// TwinCAT 3 PLC project Untitled1
// ProgramVersion: 3.1.4024.0
// libraries:
//   Tc2_Standard, * (Beckhoff Automation GmbH)
//   Tc2_System, * (Beckhoff Automation GmbH)
//   Tc3_Module, * (Beckhoff Automation GmbH)
//   VisuSymbols,3.5.10.0,System
// project tree:
//   / GlobalTextList.TcGTLO, PlcTask.TcTTO, Visualisierungsmanager.TcVMO (not stored)
//   GVLs/ GVL.TcGVL
//   POUs/ FuelMeasurement.TcPOU, MAIN.TcPOU
//   VISUs/ Visualization.TcVIS
// real-time tasks:
//   TASK PlcTask: cycle T#10ms, priority 20, ADS port 350
// I/O:
//   DEVICE Gerät 2 (CX7000), AmsNetId 5.156.235.236.3.1
//     Klemme 1 (CX7028) [CX7028-0000-0121]
//       modules: Module 1 (DIO_2x), Module 2 (Empty Module), Module 3 (DIO_2x), Module 4 (Empty Module), Module 5 (DI_2x), Module 6 (Empty Module), Module 7 (DI_2x), Module 8 (Empty Module)
// variable links:
//   Untitled1/Untitled1 Instance <-> Device 2 (CX7000)/Term 1 (CX7028)
//     PlcTask Inputs/GVL.sensorN1 <-> Module 1 (DIO_2x)/DIO_2x Input Channel 1/Input
//     PlcTask Inputs/GVL.sensorN2 <-> Module 3 (DIO_2x)/DIO_2x Input Channel 1/Input
//     PlcTask Outputs/GVL.ValveN2 <-> Module 3 (DIO_2x)/DIO_2x Output Channel 1/Output
//     PlcTask Outputs/GVL.valveN1 <-> Module 1 (DIO_2x)/DIO_2x Output Channel 1/Output

CONFIGURATION Untitled1
    RESOURCE PLC ON TwinCAT3
        TASK PlcTask(INTERVAL := T#10ms, PRIORITY := 20);
        PROGRAM MAIN WITH PlcTask : MAIN;
    END_RESOURCE
END_CONFIGURATION

// ---- GVLs/GVL.TcGVL
{attribute 'qualified_only'}
VAR_GLOBAL
	
	sensorN1 AT %I* : BOOL ;
	sensorN2 AT %I* : BOOL ;
	
	valveN1 AT %Q* : BOOL;
	ValveN2 AT %Q* : BOOL;
	
	bStartMeasurement : BOOL := FALSE;
	
	
END_VAR

// ---- POUs/MAIN.TcPOU
PROGRAM MAIN
VAR
	iCounter AT %Q*		: DINT;

	FuelMeasurement1 : FuelMeasurement;
	recordedTime : TIME ;
	bMeasurementOngoing1 : BOOL;
	valveN1 : BOOL ;
	valveN2 : BOOL ;
	FuelVolumePerSec : REAL;
	bMeasurementDone1 : BOOL := FALSE;
	
	//bMeasurementOngoing2: BOOL := FALSE;
END_VAR

iCounter := iCounter + 1;



FuelMeasurement1(bFuelMeasurement := GVL.bStartMeasurement, valveN1 => GVL.valveN1,valveN2 => GVL.ValveN2 , timeElapsed => recordedTime, bEndFB => bMeasurementDone1, FuelVolumePerSec => FuelVolumePerSec);

END_PROGRAM

// ---- POUs/FuelMeasurement.TcPOU
FUNCTION_BLOCK FuelMeasurement
VAR CONSTANT
	TankVolume : INT := 334; // The volume may vary depending on the tank volume.
	
END_VAR
VAR_INPUT
	bFuelMeasurement : BOOL := TRUE;
	
END_VAR
VAR_OUTPUT
	timeElapsed: TIME := T#0S;
	
	valveN1 : BOOL := FALSE;
	valveN2 : BOOL := FALSE;
	bEndFB : BOOL;
	FuelVolumePerSec : REAL := 0;
	
END_VAR
VAR
	bMeasurementDone : BOOL;
	readyToCount : BOOL := FALSE;
	timeStart: TIME;  
 	timerRunning: BOOL := FALSE;
	
	readyToClose : BOOL := FALSE;
	
	TimeToReal : REAL;
	//bMeasurementDone: BOOL := FALSE;
	INT1: INT :=0;
END_VAR

(*
IF GVL.sensorN1 AND GVL.sensorN2 AND bFuelMeasurement THEN
	valveN1 := TRUE;
	valveN2 := TRUE;
	readyToCount := TRUE;
END_IF  

IF NOT GVL.sensorN1 AND readyToCount THEN
	timeStart := TIME();
	readyToCount := FALSE;
	timerRunning := TRUE;
END_IF

IF NOT GVL.sensorN2 AND timerRunning THEN
	timeElapsed := TIME() - timeStart;
	timerRunning := FALSE;
	bMeasurementDone := TRUE;
END_IF

TimeToReal := (TIME_TO_REAL(timeElapsed)/ 1000); // The unit of TimeToReal is Second.
FuelVolumePerSec := TankVolume / (TimeToReal/60) ;

IF bMeasurementDone THEN
	valveN1 := FALSE;
	valveN2 := FALSE;
	bEndFB := TRUE;
END_IF
*)
(*--------------------State---------------------*)

CASE INT1 OF
0:
	IF GVL.sensorN1 AND GVL.sensorN2 THEN
		INT1 := 10;
	END_IF
10:  //Ready
	IF GVL.sensorN1 AND GVL.sensorN2 AND bFuelMeasurement THEN
	valveN1 := TRUE;
	valveN2 := TRUE;
	//readyToCount := TRUE;
	INT1 := 20;
	END_IF  
20:  //Wait for upper sensor
	IF NOT GVL.sensorN1 THEN
	timeStart := TIME();
	//readyToCount := FALSE;
	timerRunning := TRUE;
	INT1 := 30;
	END_IF   
30: //Wait for lower sensor
	IF NOT GVL.sensorN2 THEN
	timeElapsed := TIME() - timeStart;
	timerRunning := FALSE;
	//bMeasurementDone := TRUE;
	
	TimeToReal := (TIME_TO_REAL(timeElapsed)/ 1000); // The unit of TimeToReal is Second.
	FuelVolumePerSec := TankVolume / (TimeToReal/60) ;

	INT1 := 40;
	END_IF
40: //Measurement finished
	
	//IF bMeasurementDone THEN
	valveN1 := FALSE;
	valveN2 := FALSE;
	bEndFB := TRUE;
	//bMeasurementDone := FALSE;
	IF GVL.sensorN1 AND GVL.sensorN2 THEN
	INT1 := 10;
	END_IF
	
END_CASE;

END_FUNCTION_BLOCK

// ---- GlobalTextList.TcGTLO
TEXTLIST GlobalTextList
  158 = '%.2f ml/min'
  333 = '%0.1f'
  71 = 'Screen one'
  77 = 'State: %d'
END_TEXTLIST

// ---- VISUs/Visualization.TcVIS
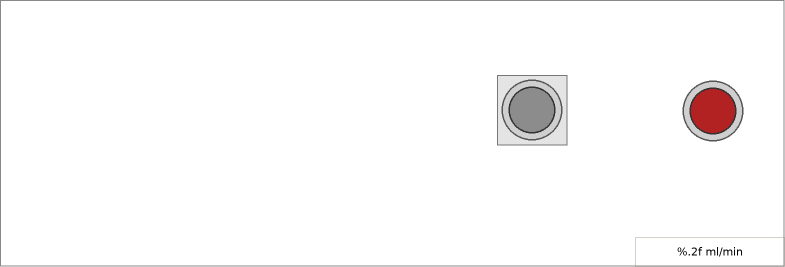
VISUALIZATION Visualization  // 785x267
    Lamp1 (678,76 70x70), variable: MAIN.FuelMeasurement1.timerRunning, style: Lamp-Lamp1-Red
    Textfield (635,237 150x30), "%.2f ml/min", text variable: MAIN.FuelVolumePerSec
    PushSwitch (497,75 70x70), variable: GVL.bStartMeasurement, behaviour: TAP, style: Switch-PushSwitch-Gray
END_VISUALIZATION
